FUNCTION_BLOCK Faults1
VAR_INPUT
END_VAR
VAR_OUTPUT
END_VAR
VAR
END_VAR

END_FUNCTION_BLOCK

(* stored: Version 1.1.0.1, ProductVersion 3.1.4024.11
   POU Faults1: Id {b31f38bf-7663-4012-8b28-87ccca645ac4}, SpecialFunc None *)
